(* IEC 61131-3 sources: MotionTestBenchMaster/Logical/30_MC/Task/Cyclic05/MC_IDLE, 3 files *)

(* ---- Cyclic.st ---- *)
PROGRAM _CYCLIC
(***** FUBs cyclic call *****)
	fbMpAlarmXListUI_Main();

	(* Hmi management *)
	tonUpdateHmiUi.PT	:= t#10s;
	tonUpdateHmiUi.IN	:= NOT xUpdateUi;
	tonUpdateHmiUi();

	stMainUIConnect.AcknowledgeAll	:= MC_InputOutput.Network.Machine.Commands.AlarmReset;

	IF tonUpdateHmiUi.Q THEN
		xUpdateUi	:= TRUE;
	END_IF

	IF xUpdateUi THEN
		IF strlen(ADR(stMainUIConnect.AlarmList.Message[uiStringCounter]))> 0 THEN
			strcpy(ADR(HMI_MC_AlarmList[uiStringCounter]),ADR(stMainUIConnect.AlarmList.Message[uiStringCounter]));
		ELSIF strlen(ADR(stMainUIConnect.AlarmList.Name[uiStringCounter]))> 0 THEN
			strcpy(ADR(HMI_MC_AlarmList[uiStringCounter]),ADR(stMainUIConnect.AlarmList.Name[uiStringCounter]));
		ELSE
			HMI_MC_AlarmList[uiStringCounter]:= '';
		END_IF

		uiStringCounter := (uiStringCounter + 1) MOD 10;

		IF uiStringCounter = 0 THEN
			xUpdateUi	:= FALSE;
		END_IF
	ELSE
		uiStringCounter	:= 0;
	END_IF
END_PROGRAM

(* ---- Init.st ---- *)
PROGRAM _INIT
	(* AlarmX UI Setup *)
	stMainAlarmSetup.AlarmListScrollWindow	:= 0;
	stMainAlarmSetup.AlarmListSize			:= 100;

	(* AlarmX UI Connect *)
	stMainUIConnect;

	(* Ui Init *)
	fbMpAlarmXListUI_Main.MpLink		:= ADR(gMainAlarmXCoreLink);
	fbMpAlarmXListUI_Main.UISetup		:= stMainAlarmSetup;
	fbMpAlarmXListUI_Main.UIConnect		:= ADR(stMainUIConnect);
	fbMpAlarmXListUI_Main.Enable		:= TRUE;
END_PROGRAM

(* ---- Variables.var ---- *)
(*Main*)
VAR
	tonUpdateHmiUi : TON;
	xUpdateUi : BOOL;
	uiStringCounter : UINT;
	stMainUIConnect : MpAlarmXListUIConnectType := (0);
	fbMpAlarmXListUI_Main : MpAlarmXListUI;
	stMainAlarmSetup : MpAlarmXListUISetupType;
END_VAR
